TYPE ST_MC_Status :
STRUCT
	
Status			: BOOL;
Done			: BOOL;
Busy			: BOOL;
Error			: BOOL;
Active			: BOOL;
CmdAborted		: BOOL;
InVelocity		: BOOL;
ErrorID			: UDINT;

END_STRUCT
END_TYPE

(* stored: Version 1.1.0.1, ProductVersion 3.1.4024.12
   DUT ST_MC_Status: Id {de65c54f-f555-40de-a1be-f3ed8c5e6a9b} *)
